// TIA Portal V20 export
TYPE "typeEm2CommandsJobInterface"
// stored: Access Published, Namespace Unit1
   STRUCT
      reqEm0ToRewind { ExternalWritable := 'False'} : Bool;
      reqEm1ToRewind { ExternalWritable := 'False'} : Bool;
      reqEm0To1LinkChg { ExternalWritable := 'False'} : Bool;
      reqEm1To0LinkChg { ExternalWritable := 'False'} : Bool;
   END_STRUCT;
END_TYPE
